TYPE ST_Event :
STRUCT
	eEventType : E_Event;
	eEventSeverity : TcEventSeverity;
	nEventIdentity : UDINT;
	sEventText : STRING(255);
	dtTimestamp : DATE_AND_TIME;
END_STRUCT
END_TYPE

(* stored: Version 1.1.0.1, ProductVersion 3.1.4024.16
   DUT ST_Event: Id {99acb789-da04-447e-b4a4-235813905dbd} *)
